// LS Electric XG5000 project: 8_29
// PLC LSPLC
// module base 0 slot 0: 입출력 모듈:XBC-DR14E (DC 24V 입력 8점, 릴레이 출력 6점)

PROGRAM NewProgram (task: 스캔 프로그램)

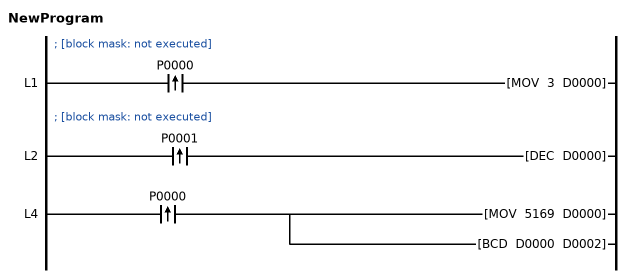
; L1 (block mask: not executed)
LOADP     P0000
MOV       3 D0000
; L2 (block mask: not executed)
LOADP     P0001
DEC       D0000
; L4
LOADP     P0000
MOV       5169 D0000
BCD       D0000 D0002